PROGRAM P_ModeSelector
VAR
	//
	// BOOL
	Mode_Power_on: BOOL;
END_VAR

//***********************************************************************************
//
// ETH Zürich / Robotic Fabrication Lab
// HIB C 13 / Stefano-Franscini-Platz 1
// CH-8093 Zürich
// 
// ***********************************************************************************
// 
// PROJECT     :  A061 Digital Casting System
// 
// FUNCTION    :  selector for mode control
// 
// AUTHOR      :  Weiting Chen
// 
// EMAIL       :  chenw@usi.ch
// 
// Copyright   :  USI , ETH Zürich (CH) 2022
//
// ***********************************************************************************


// Manual mode
GVL_VAR.b_Mode_Manual := GVL_IO.ib_CC1_Button_Mode_Manual;
 
// Laptop mode
GVL_VAR.b_Mode_Laptop := GVL_IO.ib_CC1_Button_Mode_Laptop;

// Robot mode
// Pass


IF GVL_VAR.b_Mode_Manual THEN // should be change to not 
	//
	Mode_Power_on:= GVL_IO.ib_CC1_Button_Mode_Manual;

ElSIF GVL_VAR.b_Mode_Laptop THEN
	//
	Mode_Power_on:= GVL_IO.ib_CC1_Button_Mode_Laptop;
	
END_IF

GVL_VAR.b_CC1_Mode_On:=Mode_Power_on;

END_PROGRAM

(* stored: Version 1.1.0.1, ProductVersion 3.1.4024.11
   POU P_ModeSelector: Id {0eb7d8c2-292e-4a26-bb54-34c9ce7294b6}, SpecialFunc None *)
